Universal Robots PolyScope program: orange_Wheel.urp

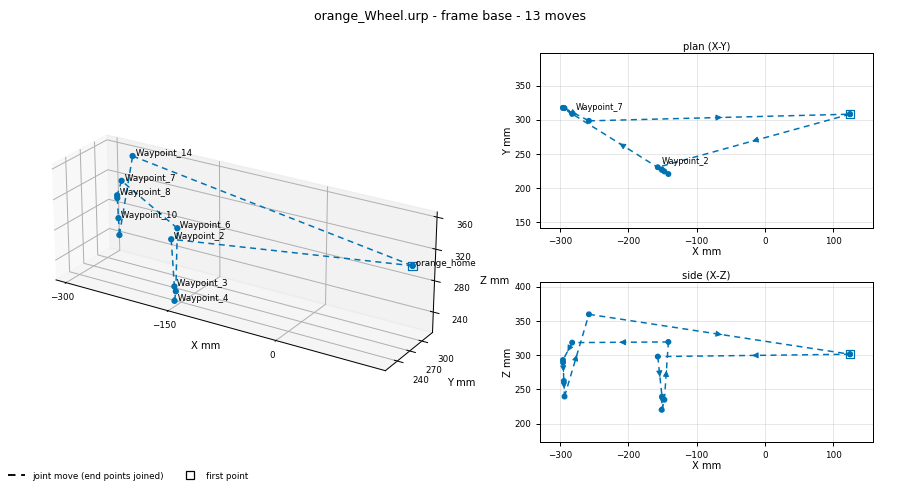
[picture p0: tool path of orange_Wheel.urp in frame base, 13 of 13 moves have a stored position in this frame; points joined in program order, loops and branches not executed]
Program orange_Wheel (installation=default directory=/programs/usbdisk/Zahra1/orangi createdIn=5.11.11.1010533 lastSavedIn=5.11.11.1010533 robotSerialNumber=20205300864)
Calibrated DH parameters: a=[-0.000166, -0.243494, -0.153108, 0.000057, -0.000123, 0]; d=[0.151897, -1.34267, 53.988124, -52.514559, 0.085283, 0.092193]; alpha=[1.572472, -0.003756, 0.002824, 1.570807, -1.572621, 0]; deltaTheta=[0, 0.020704, 7.033215, -0.770746, 0.000004, 0]
Robot Program (runOnlyOnce=true)
  MoveJ speed 60 deg/s, acceleration 80 deg/s^2 (useActiveTCP=true) feature=Base
    Waypoint orange_home: TCP in base x=124.286 y=308.277 z=301.462 mm, rx=2.2499 ry=-2.1846 rz=-0.0963 rad; joints [-269.66, -91.226, -90.279, -86.086, 92.69, 808.818] deg
    URCap Gripper (Robotiq_Grippers, Robotiq Inc.) dataModel(position=25.098039215686274, force=94.0, speed=40.0, positionInDouble=25.098039215686274, forceInDouble=94.0, speedInDouble=40.0, slaveIds=[9], blocking=true, robotCompliant=false)
    Waypoint Waypoint_2: TCP in base x=-156.913 y=230.667 z=298.044 mm, rx=-2.266 ry=2.1421 rz=0.0262 rad; joints [-207.317, -77.099, -102.98, -89.263, 88.525, 869.55] deg
    Waypoint Waypoint_3: TCP in base x=-150.735 y=226.815 z=239.491 mm, rx=-2.2808 ry=2.151 rz=0.0586 rad; joints [-207.439, -77.004, -119.59, -71.335, 89.185, 869.327] deg
    Waypoint Waypoint_4: TCP in base x=-151.181 y=227.394 z=220.152 mm, rx=-2.2808 ry=2.1511 rz=0.0586 rad; joints [-207.521, -79.007, -123.604, -65.318, 89.186, 869.263] deg
    URCap Gripper (Robotiq_Grippers, Robotiq Inc.) dataModel(position=94.41176470588235, force=94.0, speed=40.0, positionInDouble=94.41176470588235, forceInDouble=94.0, speedInDouble=40.0, slaveIds=[9], blocking=true, robotCompliant=false)
    Waypoint Waypoint_5: TCP in base x=-147.205 y=224.552 z=234.879 mm, rx=2.231 ry=-2.1859 rz=-0.1256 rad; joints [-207.517, -75.62, -123.085, -66.524, 89.619, 871.439] deg
    Waypoint Waypoint_6: TCP in base x=-141.392 y=220.749 z=319.455 mm, rx=2.2309 ry=-2.186 rz=-0.1257 rad; joints [-207.306, -71.333, -102.921, -90.97, 89.577, 871.594] deg
    Waypoint Waypoint_7: TCP in base x=-282.105 y=308.761 z=318.463 mm, rx=0.0639 ry=-3.1196 rz=-0.0236 rad; joints [-209.354, -113.958, -56.894, -97.556, 89.786, 958.364] deg
    Waypoint Waypoint_8: TCP in base x=-295.587 y=317.56 z=293.003 mm, rx=-0.0634 ry=3.0987 rz=-0.0142 rad; joints [-209.358, -119.495, -53.848, -98.903, 89.131, 958.381] deg
    Waypoint Waypoint_9: TCP in base x=-295.438 y=317.505 z=289.411 mm, rx=-0.0635 ry=3.0987 rz=-0.0143 rad; joints [-209.365, -119.343, -55.057, -97.848, 89.137, 958.373] deg
    Waypoint Waypoint_10: TCP in base x=-294.28 y=317.293 z=262.393 mm, rx=-0.0634 ry=3.0988 rz=-0.0142 rad; joints [-209.434, -118.833, -63.125, -90.284, 89.15, 958.32] deg
    Waypoint Waypoint_1: TCP in base x=-293.31 y=317.112 z=239.641 mm, rx=-0.0634 ry=3.0987 rz=-0.0143 rad; joints [-209.491, -119.127, -68.807, -84.312, 89.157, 958.277] deg
    URCap Gripper (Robotiq_Grippers, Robotiq Inc.) dataModel(position=21.176470588235293, force=70.0, speed=67.0, positionInDouble=21.176470588235293, forceInDouble=70.0, speedInDouble=67.0, slaveIds=[9], blocking=true, robotCompliant=false)
    Waypoint Waypoint_14: TCP in base x=-257.613 y=298.562 z=359.879 mm, rx=0.0615 ry=-3.076 rz=-0.1134 rad; joints [-209.409, -107.374, -56.446, -100.824, 88.118, 958.276] deg
    Waypoint orange_home: TCP in base x=124.286 y=308.277 z=301.462 mm, rx=2.2499 ry=-2.1846 rz=-0.0963 rad; joints [-269.66, -91.226, -90.279, -86.086, 92.69, 808.818] deg
